FUNCTION_BLOCK FB_CanNodeBase EXTENDS FB_HwModule
VAR_INPUT
END_VAR
VAR_OUTPUT
END_VAR
VAR
	stAdsAdress		: ST_AdsAdress;
	bNodeEnabled	: BOOL;
	bNodeFound		: BOOL;
	nNodeId			: USINT;
	nNodeState		AT %I* : USINT;	//PDO
	nErrorId 		: ERRORID;
	nErrorId2 		: UDINT;
	sHardwVersion	: STRING(15);
	sSoftwVersion	: STRING(15);
	
	bPrepare			: BOOL;
	nStateA_Prepare 	: USINT;
	bPreparingOK		: BOOL;
	
	bResetError		: BOOL;
	nStateResetError: USINT;
	
	bResetApp		: BOOL;
	nStateA_ResetApp: USINT;
	
	fbSdoRead 		: FB_SDO_READ;
	fbSdoWrite		: FB_SDO_WRITE;
	nPOUState 		: USINT;
	
	bStopMonitor	: BOOL;
	
	timeout			: TON;
END_VAR

IF bPrepare THEN
	A_Prepare();
	IF nStateA_Prepare >= 80 THEN
		IF nStateA_Prepare >= 99 THEN
			bError := TRUE;
		ELSE
			bPreparingOK := TRUE;
		END_IF
		nStateA_Prepare := 0;
		bPrepare := FALSE;
	END_IF
END_IF

IF bResetApp THEN
	A_ResetApp();
	IF nStateA_ResetApp >= 80 THEN
		IF nStateA_ResetApp >= 99 THEN
			bError := TRUE;
		END_IF
		nStateA_ResetApp := 0;
		bResetApp := FALSE;
	END_IF
END_IF

bBusy := bPrepare OR bResetError OR bResetApp;

ACTION A_Monitor:
IF nNodeState > 0  THEN
	bError := TRUE;
END_IF
END_ACTION

ACTION A_Prepare:
nPOUState := nStateA_Prepare;
CASE nStateA_Prepare OF
	0:	//Checken, ob Node "operational"
		//Timeout von 10s
		timeout(IN:= TRUE, PT:= T#10S);
		IF nNodeState = 0 THEN
			timeout(IN:= FALSE);
			bNodeFound := TRUE;
			nStateA_Prepare := 1;
		END_IF
		IF timeout.Q THEN
			timeout(IN:= FALSE);
			nStateA_Prepare := 99;
			CASE nNodeState OF
				1:	nErrorId := E_ErrorIdCan.ERRORID_NodeDeactivated;
				2:	nErrorId := E_ErrorIdCan.ERRORID_NodeNotFound;
					//Nur in Fehler gehen, wenn Node die Kopfbasisplatine ist.
					//Ein Error zu folge hätte, dann würde es auch bei einem abgestecktem Mtp-Heater zu einem Error kommen.
					IF stHardwareId.eGroup <> E_HardwareGrp.MultiZBasis THEN
						nStateA_Prepare := 80;	
					END_IF
				4:	nErrorId := E_ErrorIdCan.ERRORID_SdoSyntaxErrorAtStartup;
				5:	nErrorId := E_ErrorIdCan.ERRORID_SdoDataMismatchAtStartup;
				12:	nErrorId := E_ErrorIdCan.ERRORID_NodePreOP;
			END_CASE
		END_IF

	1:	//Hardwareversion auslesen
		fbSdoRead(sADSNetID:= stAdsAdress.sNetId, nPortNr:= stAdsAdress.nPort,
				nIndex:= 16#1009, nSubIndex:= 0, nDataLength:= 20, bExecute:= TRUE);
				
		IF NOT fbSdoRead.bBusy THEN
			IF fbSdoRead.bError THEN
				nErrorId := fbSdoRead.nAdsErrorId;
				nErrorId2 := fbSdoRead.nSdoErrorId;
				nStateA_Prepare := 99;	//Error
			ELSE
				sHardwVersion := fbSdoRead.sData;
				nStateA_Prepare := 2;
			END_IF
			fbSdoRead(bExecute:= FALSE);
		END_IF
		
	2:	//Softwareversion auslesen
		fbSdoRead(sADSNetID:= stAdsAdress.sNetId, nPortNr:= stAdsAdress.nPort,
				nIndex:= 16#100A, nSubIndex:= 0, nDataLength:= 20, bExecute:= TRUE);
				
		IF NOT fbSdoRead.bBusy THEN
			IF fbSdoRead.bError THEN
				nErrorId := fbSdoRead.nAdsErrorId;
				nErrorId2 := fbSdoRead.nSdoErrorId;
				nStateA_Prepare := 99;	//Error
			ELSE
				sSoftwVersion := fbSdoRead.sData;
				nStateA_Prepare := 80;
			END_IF
			fbSdoRead(bExecute:= FALSE);
		END_IF
	
END_CASE

IF nStateA_Prepare = 99 THEN
	stError.Cmd := 0;
	stError.ErrorId := nErrorId;
	stError.HardwareGrp := stHardwareId.eGroup;
	stError.HardwareNr := stHardwareId.nItem;
END_IF
END_ACTION

ACTION A_ResetApp:
nStateA_ResetApp := 80;
END_ACTION

METHOD M_GetHwInfo : ST_HardwareInfo
VAR_INPUT
END_VAR
M_GetHwInfo := SUPER^.M_GetHwInfo();
M_GetHwInfo.sHardwVersion := sHardwVersion;
M_GetHwInfo.sSoftwVersion := sSoftwVersion;
END_METHOD

METHOD M_Prepare
VAR_INPUT
	sAdsNetId	: STRING(23);
	nCanNodeId	: USINT;
END_VAR
stAdsAdress.sNetId := sAdsNetId;
stAdsAdress.nPort := nCanNodeId + 4096;
nNodeId := nCanNodeId;
bNodeEnabled := TRUE;
bPrepare := TRUE;
bPreparingOK := FALSE;
END_METHOD

METHOD M_Reset
VAR_INPUT
END_VAR
IF bError THEN
	bResetError := TRUE;
END_IF
END_METHOD

METHOD M_ResetApp
VAR_INPUT
END_VAR
bResetApp := TRUE;
END_METHOD

PROPERTY P_bNodeEnabled : BOOL
GET
P_bNodeEnabled := bNodeEnabled;
END_GET
END_PROPERTY

PROPERTY P_bStopMonitor : BOOL
GET
P_bStopMonitor := bStopMonitor;
END_GET
SET
bStopMonitor := P_bStopMonitor;
END_SET
END_PROPERTY

PROPERTY P_nAdsPort : UINT
GET
P_nAdsPort := stAdsAdress.nPort;
END_GET
END_PROPERTY

PROPERTY P_nNodeId : USINT
GET
P_nNodeId := nNodeId;
END_GET
END_PROPERTY

PROPERTY P_nNodeState : USINT
GET
P_nNodeState := nNodeState;
END_GET
END_PROPERTY

PROPERTY P_sAdsNetId : STRING(23)
GET
P_sAdsNetId := stAdsAdress.sNetId;
END_GET
END_PROPERTY

PROPERTY P_sHardwVersion : STRING(15)
GET
P_sHardwVersion := sHardwVersion;
END_GET
END_PROPERTY

PROPERTY P_sSoftwVersion : STRING(15)
GET
P_sSoftwVersion := sSoftwVersion;
END_GET
END_PROPERTY

END_FUNCTION_BLOCK

(* stored: Version 1.1.0.1, ProductVersion 3.1.4024.11
   POU FB_CanNodeBase: Id {b9ec44d1-32d5-48f9-a4be-3244e9a62111}, SpecialFunc None
   Action A_Monitor: Id {0d17c58a-e01a-445a-b762-2a34737c732c}
   Action A_Prepare: Id {03af6d06-3a0c-44ed-993d-f1f04445b64e}
   Action A_ResetApp: Id {b4df81c7-2860-4bb6-a757-1bd4c4080877}
   Method M_GetHwInfo: Id {e2728c97-1dcc-42b0-979f-0bc23b688b75}
   Method M_Prepare: Id {df7aae7f-708a-49a0-8cbb-d2dc76284000}
   Method M_Reset: Id {3b4e5415-444f-40fb-a667-87fc7eaa3528}
   Method M_ResetApp: Id {a5af6c9b-c604-4312-87b5-76ce3df628fe}
   Property P_bNodeEnabled: Id {0e66fe84-7f28-448f-b8b7-3036158be19b}
   Get Get: Id {83680e29-40e1-435a-b057-300f15522e47}
   Property P_bStopMonitor: Id {45874c62-3dcb-440e-8649-e785d11e48d7}
   Get Get: Id {98a02e4d-9bc8-4c3a-8d11-0e234e12a4c6}
   Set Set: Id {c93449ed-8e7b-4cdb-8f64-1a80ca7b78a9}
   Property P_nAdsPort: Id {6848950f-a1d2-45d3-bf84-b343725deeda}
   Get Get: Id {4a86aa97-c218-41cc-9a6d-25cc62dbe0a6}
   Property P_nNodeId: Id {dcdb7a94-7c75-4152-ae3d-d6d003a4662e}
   Get Get: Id {d6b8713a-f10b-4a04-a227-0d991c9bdfc1}
   Property P_nNodeState: Id {ea850228-3a02-41d0-866d-57183016bb1d}
   Get Get: Id {53bb4b89-dc9b-468d-9670-603647029f44}
   Property P_sAdsNetId: Id {e6993480-e908-4873-8799-19c59dcf1739}
   Get Get: Id {94ea743a-2ee8-4b31-8720-a6eb4ae758ef}
   Property P_sHardwVersion: Id {cc66ad82-59a6-4382-ab33-643e32dbc3d6}
   Get Get: Id {17eb6615-83b1-4be4-a762-24a136099fcf}
   Property P_sSoftwVersion: Id {be680b16-59ae-46ef-9977-f01a860632b4}
   Get Get: Id {edbb4a38-166c-4d2e-ab51-c829415f9008} *)
